{attribute 'qualified_only'}
{attribute 'strict'}
TYPE E_SPEED_TYPE :
(
	MM_PER_SECOND,
  PERCENT
);
END_TYPE

(* stored: Version 1.1.0.1, ProductVersion 3.1.4024.12
   DUT E_SPEED_TYPE: Id {a810dcdb-df25-4ab0-b836-1bdcce2c0df6} *)
